# EPICS autosave request: CARSApp/Db/GSE_CD_MonoPositions_settings.req
$(P)$(MONO):MonoPosition
$(P)$(MONO):Mono111ThetaOffset
$(P)$(MONO):Mono311ThetaOffset
$(P)$(MONO):Mono111HeightOffset
$(P)$(MONO):Mono311HeightOffset
$(P)$(MONO):Mono111Pitch
$(P)$(MONO):Mono311Pitch
$(P)$(MONO):Mono111Roll
$(P)$(MONO):Mono311Roll
$(P)$(MONO):Mono111DSpace
$(P)$(MONO):Mono311DSpace
